TYPE ST_CounterControlOut :
STRUCT
	stButtonSave		: ST_HMI_BUTTON_OUT;
	stButtonReset		: ST_HMI_BUTTON_OUT;		
	bVisible_UserLevel	: BOOL;
	nUserLevelUsers		: INT; //count of recipe mode list
	aUserLevelUsers		: ARRAY[0..E_User_Level.eUser_Level_nMaxIdx] OF ST_Text;
	bVisible_Reaction	: BOOL;
	nReaction			: INT; //count of recipe mode list
	aReaction			: ARRAY[0..E_CounterReaction.eCounterReaction_Max] OF ST_Text;	
	bVisible_Number		: BOOL;
	bVisible_String		: BOOL;
	bVisibleInfo		: BOOL;
	stInfo				: ST_Text;
END_STRUCT
END_TYPE

(* stored: Version 1.1.0.1, ProductVersion 3.1.4024.12
   DUT ST_CounterControlOut: Id {2dff2447-1788-414a-a5d0-ac7883e9eccb} *)
